{attribute 'qualified_only'}
{attribute 'strict'}
TYPE ProfileJerkSignsEnum :
(
	uddu,
  udud 
);
END_TYPE

(* stored: Version 1.1.0.1, ProductVersion 3.1.4024.6
   DUT ProfileJerkSignsEnum: Id {b8a5c43f-13de-4042-9633-9e96e9516e46} *)
